INTERFACE I_ListComponent

METHOD PUBLIC M_Add : BOOL
VAR_INPUT
	Object: 	I_Component;
END_VAR
END_METHOD

METHOD PUBLIC M_Clear : BOOL
END_METHOD

METHOD PUBLIC M_Find : DINT
VAR_INPUT
	Object: 	I_Component;
END_VAR
END_METHOD

METHOD PUBLIC M_Index : I_Component
VAR_INPUT
	Index: 	DINT;
END_VAR
END_METHOD

METHOD PUBLIC M_Remove : BOOL
VAR_INPUT
	Object: 	I_Component;
END_VAR
END_METHOD

METHOD PUBLIC M_Request : BOOL
VAR_INPUT
	eRequest:		E_Request;
END_VAR
END_METHOD

PROPERTY P_Length : DINT
GET
END_GET
END_PROPERTY

END_INTERFACE

(* stored: Version 1.1.0.1
   Itf I_ListComponent: Id {ab8205a2-82ac-4799-980f-541526123c48}
   Method M_Add: Id {31416f6e-5c2d-4ce2-873c-dc73b1cfa758}
   Method M_Clear: Id {bec35183-59fd-4e05-8c88-04323521ec68}
   Method M_Find: Id {9f020047-7fe7-44c3-b7ac-d3f89fe85683}
   Method M_Index: Id {aa739692-a960-4472-8c48-c3bba57fc92f}
   Method M_Remove: Id {6961a1f7-e686-48a7-b56a-c7aec47523ba}
   Method M_Request: Id {92387029-bdad-43b6-9627-c14b089e9780}
   Property P_Length: Id {49615258-7cc8-4370-999e-56e1024f4c79}
   Get Get: Id {ec48dc05-e74e-4cfe-acf2-317ea9ff6055} *)
